(* IEC 61131-3 sources: tesi_iac_openplc/example, 1 file *)

(* ---- demo.st ---- *)
PROGRAM demo
  VAR
    PB1 AT %IX100.0 : BOOL;
    PB2 AT %IX100.1 : BOOL;
    LED AT %QX100.0 : BOOL;
  END_VAR

  LED := NOT(PB2) AND (LED OR PB1);
END_PROGRAM

CONFIGURATION Config0

  RESOURCE Res0 ON PLC
    TASK task0(INTERVAL := T#20ms,PRIORITY := 0);
    PROGRAM instance0 WITH task0 : demo;
  END_RESOURCE
END_CONFIGURATION
